TYPE E_MonthPL :(Stycznen:=1, Luty, Marzec, Kwiecien, Maj,  Czerwiec, Lipiec, Sierpien, Wrzesien, Pazdziernik, Listopad, Grudzien);
END_TYPE

(* stored: Version 1.1.0.1, ProductVersion 3.1.4019.2
   DUT E_MonthPL: Id {e79eec56-37ff-4eb4-bc9e-4bcb58b66887} *)
